// TIA Portal V19 export
DATA_BLOCK "iDB_ExportFlatCtrlR1"   // DB714
// stored: AutoNumber false, InstanceOfName RecipeExport_SFB, OfSystemLibElement RecipeExport, OfSystemLibVersion 1.2
"RecipeExport_SFB"
   // VAR_INPUT
   //    REQ : Bool;
   // END_VAR
   // VAR_OUTPUT
   //    DONE : Bool;
   //    BUSY : Bool;
   //    ERROR : Bool;
   //    STATUS : Word;
   // END_VAR
   // VAR_IN_OUT
   //    RECIPE_DB : Variant;
   // END_VAR
BEGIN
END_DATA_BLOCK
